FUNCTION_BLOCK FB_TOR_CB EXTENDS FB_TOR_Base
//////////////////
//  Door sensor system . State = True >> Door Closed .
//////////////////

VAR_INPUT PERSISTENT
	// Parameters of the Object (instance/model specific) 
		
		
END_VAR

VAR_OUTPUT
	//Child objects
	
END_VAR

VAR_INPUT
	// I/O Inputs 		                                     				
		
END_VAR

VAR
	//M_ALARMMANAGEMENT VARIABLES//
		
MesDataExd			: TOR_Standard ;  

	
END_VAR

END_FUNCTION_BLOCK

(* stored: Version 1.1.0.1, ProductVersion 3.1.4024.6
   POU FB_TOR_CB: Id {458e1c02-4479-4190-985f-d7ff6eca70f8}, SpecialFunc None *)
